TYPE ST_PositionState :
(**************************************************************************************
 * 	Application		:	BoxControl Framework
 *	Revision		:	$Revision: 404529 $
 *	Revision date	:	$Date: 2018-04-23 08:21:38 +0200 (Mo., 23 Apr 2018) $
 *	Last changed by	:	$Author: b7bolm $
 *	URL				:	$URL: http://almscdc.swisslog.com/repo/SWPD/Development/BoxControlFramework/20_Release/trunk/01_Software/BCF/BCF/JumpStart/20_Product/10_App/10_Base/10_Lib/01_DUTs/ST_PositionState.TcDUT $
 *
 *	Purpose			:	Position state
 *
 * ------------------------------------------------------------------------------------
 *	Copyright Swisslog [IP AG], Switzerland. All rights reserved.
 * 
 * ------------------------------------------------------------------------------------
 *	
 * 	Revision History: 
 *
 * 	VERSION			DATE			INITIALS			DESCRIPTION
 *	0.1				01.01.2001		swl					Example
 *
 **************************************************************************************)	
STRUCT
	eMode			: E_PositionMode; // Mode of the group 
	eState 			: E_PositionState; // State of the group 
	eLastState		: E_PositionState; // Previous state of the group 
	Info			: ST_PositionInfo; // Position info
	InitRelease		: ST_InitRelease; // Release to init 
END_STRUCT
END_TYPE

(* stored: Version 1.1.0.1, ProductVersion 3.1.4022.12
   DUT ST_PositionState: Id {d0f7292b-7a51-4f54-9e8d-1f084579000e} *)
